// TIA Portal V18 export
ORGANIZATION_BLOCK "Work"   // OB123, LAD, ProgramCycle
TITLE = "Main Program Sweep (Cycle)"
{ S7_Optimized_Access := 'TRUE' }
VERSION : 0.1
// stored: AutoNumber true, IsIECCheckEnabled false, SetENOAutomatically false
   VAR_INPUT
      Initial_Call : Bool;   // Initial call of this OB
      Remanence : Bool;   // =True, if remanent data are available
   END_VAR
BEGIN

REGION Network 1: Active machine
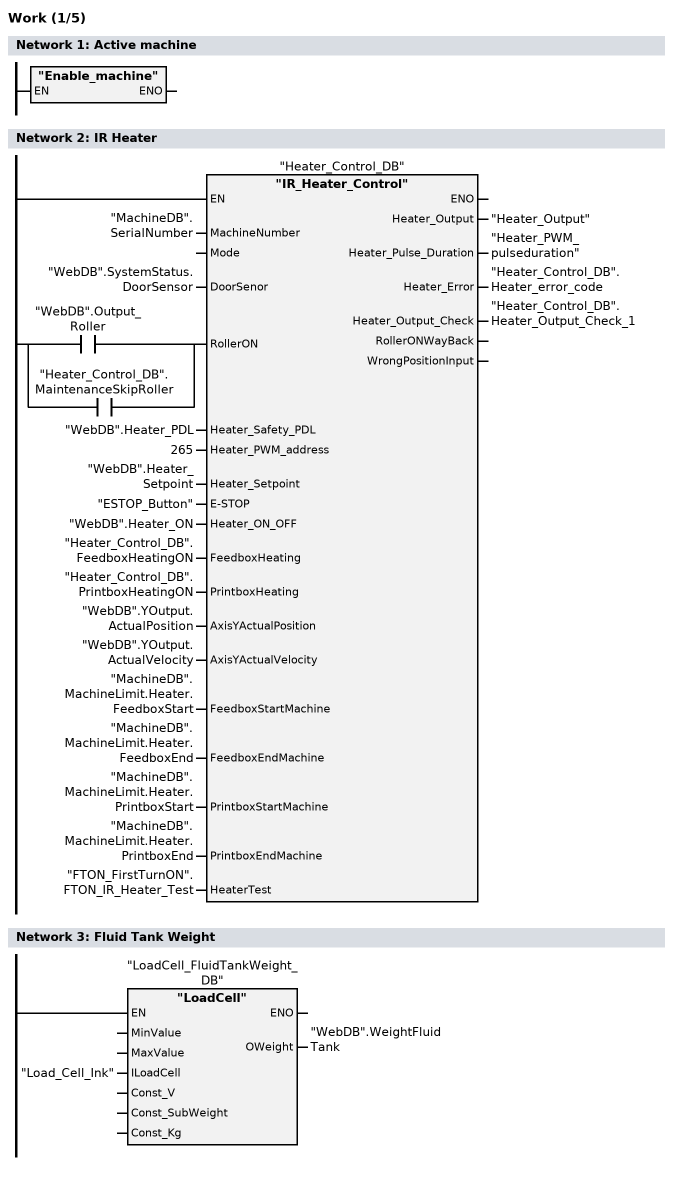
   RUNG wire#powerrail
      "Enable_machine"()
   END_RUNG
   // the same network as SCL:
   "Enable_machine"();
END_REGION

REGION Network 2: IR Heater
   RUNG wire#powerrail
      "Heater_Control_DB"(RollerON := wire#w1, MachineNumber := "MachineDB".SerialNumber, Mode :=, DoorSenor := "WebDB".SystemStatus.DoorSensor, Heater_Safety_PDL := "WebDB".Heater_PDL, Heater_PWM_address := 265, Heater_Setpoint := "WebDB".Heater_Setpoint, "E-STOP" := "ESTOP_Button", Heater_ON_OFF := "WebDB".Heater_ON, FeedboxHeating := "Heater_Control_DB".FeedboxHeatingON, PrintboxHeating := "Heater_Control_DB".PrintboxHeatingON, AxisYActualPosition := "WebDB".YOutput.ActualPosition, AxisYActualVelocity := "WebDB".YOutput.ActualVelocity, FeedboxStartMachine := "MachineDB".MachineLimit.Heater.FeedboxStart, FeedboxEndMachine := "MachineDB".MachineLimit.Heater.FeedboxEnd, PrintboxStartMachine := "MachineDB".MachineLimit.Heater.PrintboxStart, PrintboxEndMachine := "MachineDB".MachineLimit.Heater.PrintboxEnd, HeaterTest := "FTON_FirstTurnON".FTON_IR_Heater_Test, Heater_Output => "Heater_Output", Heater_Pulse_Duration => "Heater_PWM_pulseduration", Heater_Error => "Heater_Control_DB".Heater_error_code, Heater_Output_Check => "Heater_Control_DB".Heater_Output_Check_1, RollerONWayBack =>, WrongPositionInput =>)
   END_RUNG
   RUNG wire#powerrail
      Contact( "WebDB".Output_Roller )
   END_RUNG wire#w1
   RUNG wire#powerrail
      Contact( "Heater_Control_DB".MaintenanceSkipRoller )
   END_RUNG wire#w1
   // the same network as SCL:
   "Heater_Control_DB"(MachineNumber := "MachineDB".SerialNumber,   // "IR_Heater_Control"
                       DoorSenor := "WebDB".SystemStatus.DoorSensor,
                       RollerON := "WebDB".Output_Roller OR "Heater_Control_DB".MaintenanceSkipRoller,
                       Heater_Safety_PDL := "WebDB".Heater_PDL,
                       Heater_PWM_address := 265,
                       Heater_Setpoint := "WebDB".Heater_Setpoint,
                       "E-STOP" := "ESTOP_Button",
                       Heater_ON_OFF := "WebDB".Heater_ON,
                       FeedboxHeating := "Heater_Control_DB".FeedboxHeatingON,
                       PrintboxHeating := "Heater_Control_DB".PrintboxHeatingON,
                       AxisYActualPosition := "WebDB".YOutput.ActualPosition,
                       AxisYActualVelocity := "WebDB".YOutput.ActualVelocity,
                       FeedboxStartMachine := "MachineDB".MachineLimit.Heater.FeedboxStart,
                       FeedboxEndMachine := "MachineDB".MachineLimit.Heater.FeedboxEnd,
                       PrintboxStartMachine := "MachineDB".MachineLimit.Heater.PrintboxStart,
                       PrintboxEndMachine := "MachineDB".MachineLimit.Heater.PrintboxEnd,
                       HeaterTest := "FTON_FirstTurnON".FTON_IR_Heater_Test,
                       Heater_Output => "Heater_Output",
                       Heater_Pulse_Duration => "Heater_PWM_pulseduration",
                       Heater_Error => "Heater_Control_DB".Heater_error_code,
                       Heater_Output_Check => "Heater_Control_DB".Heater_Output_Check_1);
END_REGION

REGION Network 3: Fluid Tank Weight
   RUNG wire#powerrail
      "LoadCell_FluidTankWeight_DB"(MinValue :=, MaxValue :=, ILoadCell := "Load_Cell_Ink", Const_V :=, Const_SubWeight :=, Const_Kg :=, OWeight => "WebDB".WeightFluidTank)
   END_RUNG
   // the same network as SCL:
   "LoadCell_FluidTankWeight_DB"(ILoadCell := "Load_Cell_Ink", OWeight => "WebDB".WeightFluidTank);   // "LoadCell"
END_REGION

REGION Network 4: Fluid Waste Weight
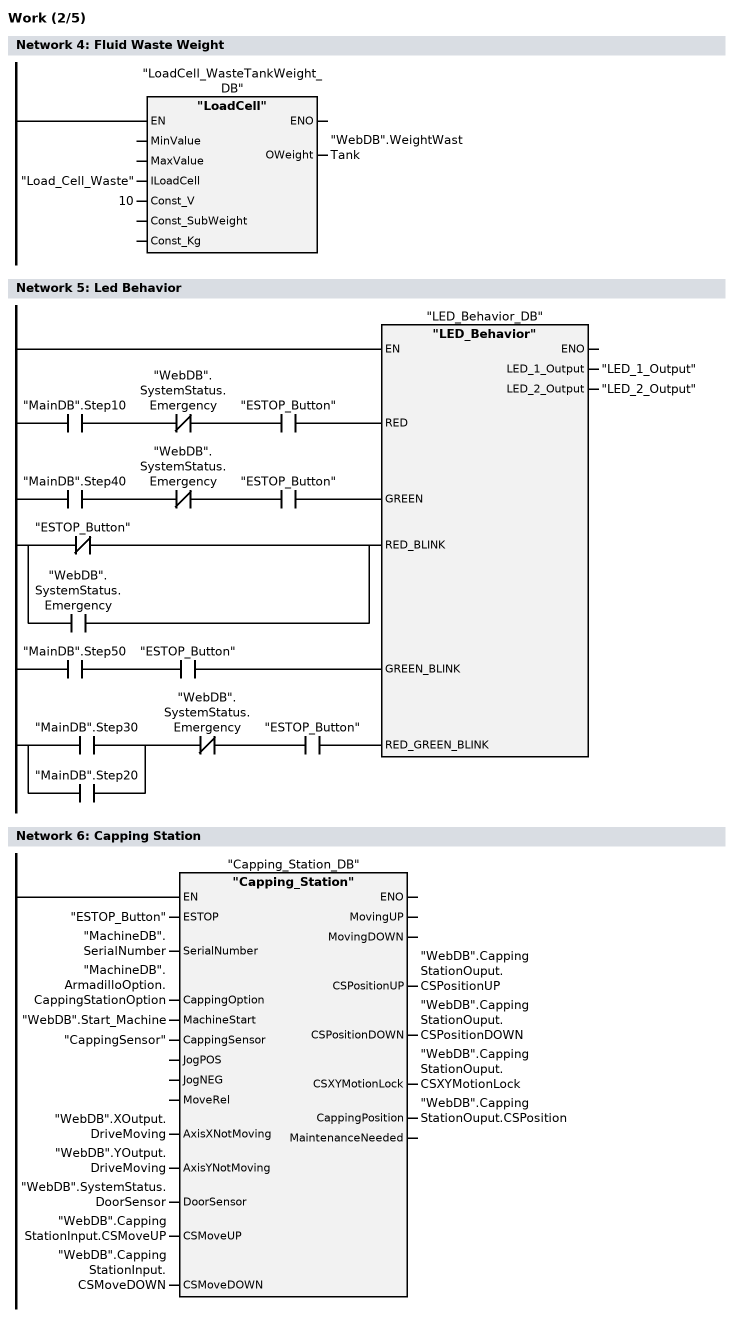
   RUNG wire#powerrail
      "LoadCell_WasteTankWeight_DB"(MinValue :=, MaxValue :=, ILoadCell := "Load_Cell_Waste", Const_V := 10, Const_SubWeight :=, Const_Kg :=, OWeight => "WebDB".WeightWastTank)
   END_RUNG
   // the same network as SCL:
   "LoadCell_WasteTankWeight_DB"(ILoadCell := "Load_Cell_Waste",   // "LoadCell"
                           Const_V := 10,
                           OWeight => "WebDB".WeightWastTank);
END_REGION

REGION Network 5: Led Behavior
   RUNG wire#powerrail
      "LED_Behavior_DB"(RED := wire#w1, GREEN := wire#w2, RED_BLINK := wire#w3, GREEN_BLINK := wire#w4, RED_GREEN_BLINK := wire#w6, LED_1_Output => "LED_1_Output", LED_2_Output => "LED_2_Output")
   END_RUNG
   RUNG wire#powerrail
      Contact( "MainDB".Step10 )
      I_Contact( "WebDB".SystemStatus.Emergency )
      Contact( "ESTOP_Button" )
   END_RUNG wire#w1
   RUNG wire#powerrail
      Contact( "MainDB".Step40 )
      I_Contact( "WebDB".SystemStatus.Emergency )
      Contact( "ESTOP_Button" )
   END_RUNG wire#w2
   RUNG wire#powerrail
      I_Contact( "ESTOP_Button" )
   END_RUNG wire#w3
   RUNG wire#powerrail
      Contact( "WebDB".SystemStatus.Emergency )
   END_RUNG wire#w3
   RUNG wire#powerrail
      Contact( "MainDB".Step50 )
      Contact( "ESTOP_Button" )
   END_RUNG wire#w4
   RUNG wire#powerrail
      Contact( "MainDB".Step30 )
      wire#w5
      I_Contact( "WebDB".SystemStatus.Emergency )
      Contact( "ESTOP_Button" )
   END_RUNG wire#w6
   RUNG wire#powerrail
      Contact( "MainDB".Step20 )
   END_RUNG wire#w5
   // the same network as SCL:
   "LED_Behavior_DB"(RED := "MainDB".Step10 AND NOT "WebDB".SystemStatus.Emergency AND "ESTOP_Button",   // "LED_Behavior"
                     GREEN := "MainDB".Step40 AND NOT "WebDB".SystemStatus.Emergency AND "ESTOP_Button",
                     RED_BLINK := NOT "ESTOP_Button" OR "WebDB".SystemStatus.Emergency,
                     GREEN_BLINK := "MainDB".Step50 AND "ESTOP_Button",
                     RED_GREEN_BLINK := ("MainDB".Step30 OR "MainDB".Step20) AND NOT "WebDB".SystemStatus.Emergency AND "ESTOP_Button",
                     LED_1_Output => "LED_1_Output",
                     LED_2_Output => "LED_2_Output");
END_REGION

REGION Network 6: Capping Station
   RUNG wire#powerrail
      "Capping_Station_DB"(ESTOP := "ESTOP_Button", SerialNumber := "MachineDB".SerialNumber, CappingOption := "MachineDB".ArmadilloOption.CappingStationOption, MachineStart := "WebDB".Start_Machine, CappingSensor := "CappingSensor", JogPOS :=, JogNEG :=, MoveRel :=, AxisXNotMoving := "WebDB".XOutput.DriveMoving, AxisYNotMoving := "WebDB".YOutput.DriveMoving, DoorSensor := "WebDB".SystemStatus.DoorSensor, CSMoveUP := "WebDB".CappingStationInput.CSMoveUP, CSMoveDOWN := "WebDB".CappingStationInput.CSMoveDOWN, MovingUP =>, MovingDOWN =>, CSPositionUP => "WebDB".CappingStationOuput.CSPositionUP, CSPositionDOWN => "WebDB".CappingStationOuput.CSPositionDOWN, CSXYMotionLock => "WebDB".CappingStationOuput.CSXYMotionLock, CappingPosition => "WebDB".CappingStationOuput.CSPosition, MaintenanceNeeded =>)
   END_RUNG
   // the same network as SCL:
   "Capping_Station_DB"(ESTOP := "ESTOP_Button",   // "Capping_Station"
                        SerialNumber := "MachineDB".SerialNumber,
                        CappingOption := "MachineDB".ArmadilloOption.CappingStationOption,
                        MachineStart := "WebDB".Start_Machine,
                        CappingSensor := "CappingSensor",
                        AxisXNotMoving := "WebDB".XOutput.DriveMoving,
                        AxisYNotMoving := "WebDB".YOutput.DriveMoving,
                        DoorSensor := "WebDB".SystemStatus.DoorSensor,
                        CSMoveUP := "WebDB".CappingStationInput.CSMoveUP,
                        CSMoveDOWN := "WebDB".CappingStationInput.CSMoveDOWN,
                        CSPositionUP => "WebDB".CappingStationOuput.CSPositionUP,
                        CSPositionDOWN => "WebDB".CappingStationOuput.CSPositionDOWN,
                        CSXYMotionLock => "WebDB".CappingStationOuput.CSXYMotionLock,
                        CappingPosition => "WebDB".CappingStationOuput.CSPosition);
END_REGION

REGION Network 7: Initial Test Sequence
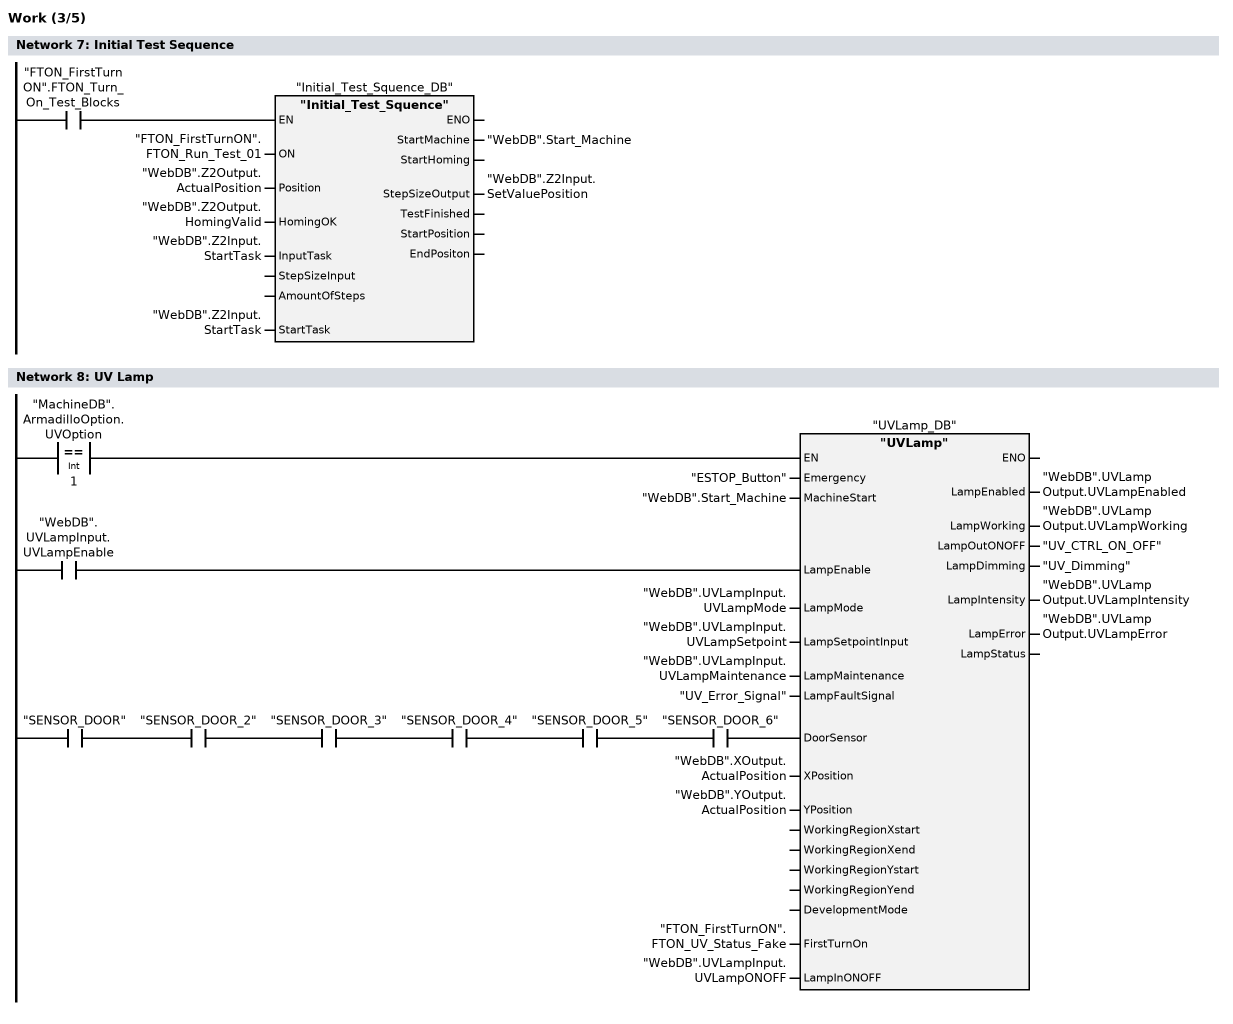
   RUNG wire#powerrail
      Contact( "FTON_FirstTurnON".FTON_Turn_On_Test_Blocks )
      "Initial_Test_Squence_DB"(ON := "FTON_FirstTurnON".FTON_Run_Test_01, Position := "WebDB".Z2Output.ActualPosition, HomingOK := "WebDB".Z2Output.HomingValid, InputTask := "WebDB".Z2Input.StartTask, StepSizeInput :=, AmountOfSteps :=, StartTask := "WebDB".Z2Input.StartTask, StartMachine => "WebDB".Start_Machine, StartHoming =>, StepSizeOutput => "WebDB".Z2Input.SetValuePosition, TestFinished =>, StartPosition =>, EndPositon =>)
   END_RUNG
   // the same network as SCL:
   IF "FTON_FirstTurnON".FTON_Turn_On_Test_Blocks THEN
       "Initial_Test_Squence_DB"(ON := "FTON_FirstTurnON".FTON_Run_Test_01,   // "Initial_Test_Squence"
                               Position := "WebDB".Z2Output.ActualPosition,
                               HomingOK := "WebDB".Z2Output.HomingValid,
                               InputTask := "WebDB".Z2Input.StartTask,
                               StartTask := "WebDB".Z2Input.StartTask,
                               StartMachine => "WebDB".Start_Machine,
                               StepSizeOutput => "WebDB".Z2Input.SetValuePosition);
   END_IF;
END_REGION

REGION Network 8: UV Lamp
   RUNG wire#powerrail
      { S7_Templates := "SrcType := Int" } EQ_Contact(in1 := "MachineDB".ArmadilloOption.UVOption, in2 := 1)
      "UVLamp_DB"(LampEnable := wire#w1, DoorSensor := wire#w2, Emergency := "ESTOP_Button", MachineStart := "WebDB".Start_Machine, LampMode := "WebDB".UVLampInput.UVLampMode, LampSetpointInput := "WebDB".UVLampInput.UVLampSetpoint, LampMaintenance := "WebDB".UVLampInput.UVLampMaintenance, LampFaultSignal := "UV_Error_Signal", XPosition := "WebDB".XOutput.ActualPosition, YPosition := "WebDB".YOutput.ActualPosition, WorkingRegionXstart :=, WorkingRegionXend :=, WorkingRegionYstart :=, WorkingRegionYend :=, DevelopmentMode :=, FirstTurnOn := "FTON_FirstTurnON".FTON_UV_Status_Fake, LampInONOFF := "WebDB".UVLampInput.UVLampONOFF, LampEnabled => "WebDB".UVLampOutput.UVLampEnabled, LampWorking => "WebDB".UVLampOutput.UVLampWorking, LampOutONOFF => "UV_CTRL_ON_OFF", LampDimming => "UV_Dimming", LampIntensity => "WebDB".UVLampOutput.UVLampIntensity, LampError => "WebDB".UVLampOutput.UVLampError, LampStatus =>)
   END_RUNG
   RUNG wire#powerrail
      Contact( "WebDB".UVLampInput.UVLampEnable )
   END_RUNG wire#w1
   RUNG wire#powerrail
      Contact( "SENSOR_DOOR" )
      Contact( "SENSOR_DOOR_2" )
      Contact( "SENSOR_DOOR_3" )
      Contact( "SENSOR_DOOR_4" )
      Contact( "SENSOR_DOOR_5" )
      Contact( "SENSOR_DOOR_6" )
   END_RUNG wire#w2
   // the same network as SCL:
   IF "MachineDB".ArmadilloOption.UVOption = 1 THEN
       "UVLamp_DB"(Emergency := "ESTOP_Button",   // "UVLamp"
                   MachineStart := "WebDB".Start_Machine,
                   LampEnable := "WebDB".UVLampInput.UVLampEnable,
                   LampMode := "WebDB".UVLampInput.UVLampMode,
                   LampSetpointInput := "WebDB".UVLampInput.UVLampSetpoint,
                   LampMaintenance := "WebDB".UVLampInput.UVLampMaintenance,
                   LampFaultSignal := "UV_Error_Signal",
                   DoorSensor := "SENSOR_DOOR" AND "SENSOR_DOOR_2" AND "SENSOR_DOOR_3" AND "SENSOR_DOOR_4" AND "SENSOR_DOOR_5" AND "SENSOR_DOOR_6",
                   XPosition := "WebDB".XOutput.ActualPosition,
                   YPosition := "WebDB".YOutput.ActualPosition,
                   FirstTurnOn := "FTON_FirstTurnON".FTON_UV_Status_Fake,
                   LampInONOFF := "WebDB".UVLampInput.UVLampONOFF,
                   LampEnabled => "WebDB".UVLampOutput.UVLampEnabled,
                   LampWorking => "WebDB".UVLampOutput.UVLampWorking,
                   LampOutONOFF => "UV_CTRL_ON_OFF",
                   LampDimming => "UV_Dimming",
                   LampIntensity => "WebDB".UVLampOutput.UVLampIntensity,
                   LampError => "WebDB".UVLampOutput.UVLampError);
   END_IF;
END_REGION

REGION Network 9: Stacklight
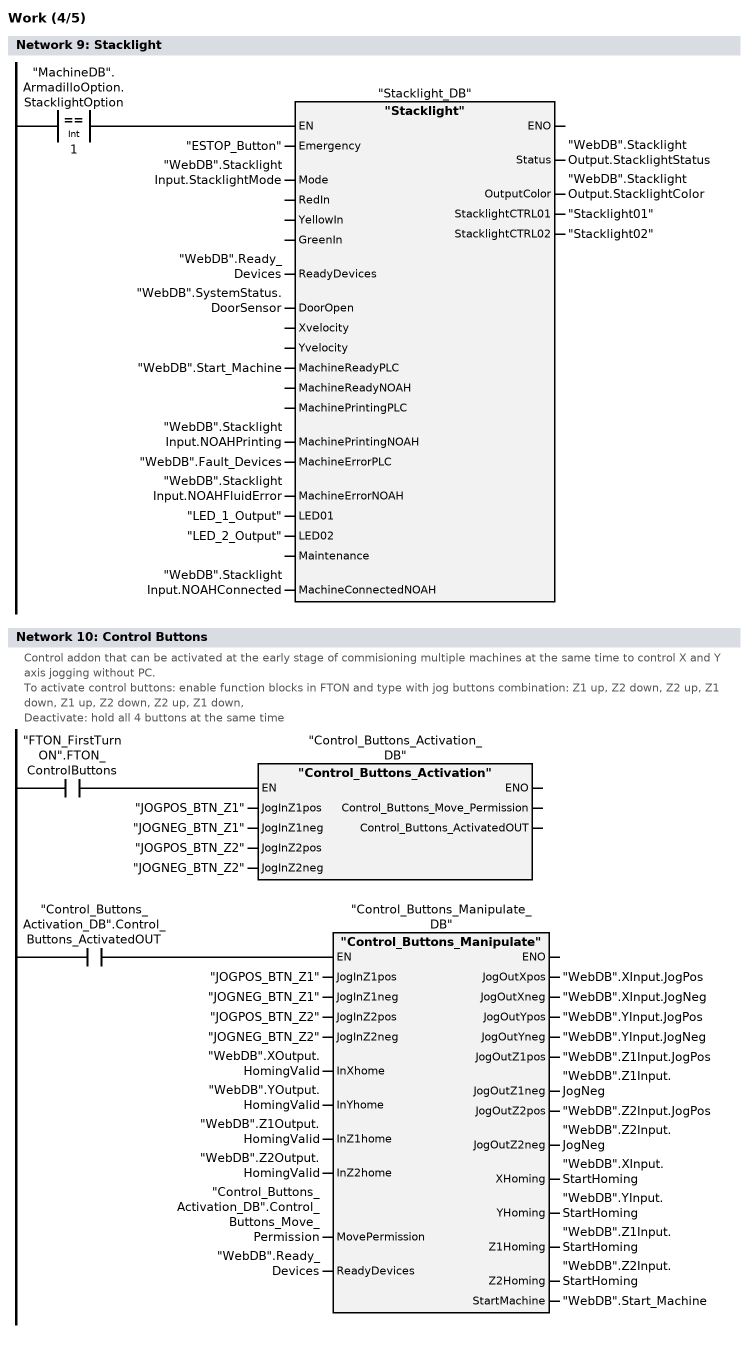
   RUNG wire#powerrail
      { S7_Templates := "SrcType := Int" } EQ_Contact(in1 := "MachineDB".ArmadilloOption.StacklightOption, in2 := 1)
      "Stacklight_DB"(Emergency := "ESTOP_Button", Mode := "WebDB".StacklightInput.StacklightMode, RedIn :=, YellowIn :=, GreenIn :=, ReadyDevices := "WebDB".Ready_Devices, DoorOpen := "WebDB".SystemStatus.DoorSensor, Xvelocity :=, Yvelocity :=, MachineReadyPLC := "WebDB".Start_Machine, MachineReadyNOAH :=, MachinePrintingPLC :=, MachinePrintingNOAH := "WebDB".StacklightInput.NOAHPrinting, MachineErrorPLC := "WebDB".Fault_Devices, MachineErrorNOAH := "WebDB".StacklightInput.NOAHFluidError, LED01 := "LED_1_Output", LED02 := "LED_2_Output", Maintenance :=, MachineConnectedNOAH := "WebDB".StacklightInput.NOAHConnected, Status => "WebDB".StacklightOutput.StacklightStatus, OutputColor => "WebDB".StacklightOutput.StacklightColor, StacklightCTRL01 => "Stacklight01", StacklightCTRL02 => "Stacklight02")
   END_RUNG
   // the same network as SCL:
   IF "MachineDB".ArmadilloOption.StacklightOption = 1 THEN
       "Stacklight_DB"(Emergency := "ESTOP_Button",   // "Stacklight"
                       Mode := "WebDB".StacklightInput.StacklightMode,
                       ReadyDevices := "WebDB".Ready_Devices,
                       DoorOpen := "WebDB".SystemStatus.DoorSensor,
                       MachineReadyPLC := "WebDB".Start_Machine,
                       MachinePrintingNOAH := "WebDB".StacklightInput.NOAHPrinting,
                       MachineErrorPLC := "WebDB".Fault_Devices,
                       MachineErrorNOAH := "WebDB".StacklightInput.NOAHFluidError,
                       LED01 := "LED_1_Output",
                       LED02 := "LED_2_Output",
                       MachineConnectedNOAH := "WebDB".StacklightInput.NOAHConnected,
                       Status => "WebDB".StacklightOutput.StacklightStatus,
                       OutputColor => "WebDB".StacklightOutput.StacklightColor,
                       StacklightCTRL01 => "Stacklight01",
                       StacklightCTRL02 => "Stacklight02");
   END_IF;
END_REGION

REGION Network 10: Control Buttons
   // Control addon that can be activated at the early stage of commisioning multiple machines at the same time to control X and Y axis jogging without PC.
   // 
   // To activate control buttons: enable function blocks in FTON and type with jog buttons combination: Z1 up, Z2 down, Z2 up, Z1 down, Z1 up, Z2 down, Z2 up, Z1 down,
   // 
   // Deactivate: hold all 4 buttons at the same time
   RUNG wire#powerrail
      Contact( "FTON_FirstTurnON".FTON_ControlButtons )
      "Control_Buttons_Activation_DB"(JogInZ1pos := "JOGPOS_BTN_Z1", JogInZ1neg := "JOGNEG_BTN_Z1", JogInZ2pos := "JOGPOS_BTN_Z2", JogInZ2neg := "JOGNEG_BTN_Z2", Control_Buttons_Move_Permission =>, Control_Buttons_ActivatedOUT =>)
   END_RUNG
   RUNG wire#powerrail
      Contact( "Control_Buttons_Activation_DB".Control_Buttons_ActivatedOUT )
      "Control_Buttons_Manipulate_DB"(JogInZ1pos := "JOGPOS_BTN_Z1", JogInZ1neg := "JOGNEG_BTN_Z1", JogInZ2pos := "JOGPOS_BTN_Z2", JogInZ2neg := "JOGNEG_BTN_Z2", InXhome := "WebDB".XOutput.HomingValid, InYhome := "WebDB".YOutput.HomingValid, InZ1home := "WebDB".Z1Output.HomingValid, InZ2home := "WebDB".Z2Output.HomingValid, MovePermission := "Control_Buttons_Activation_DB".Control_Buttons_Move_Permission, ReadyDevices := "WebDB".Ready_Devices, JogOutXpos => "WebDB".XInput.JogPos, JogOutXneg => "WebDB".XInput.JogNeg, JogOutYpos => "WebDB".YInput.JogPos, JogOutYneg => "WebDB".YInput.JogNeg, JogOutZ1pos => "WebDB".Z1Input.JogPos, JogOutZ1neg => "WebDB".Z1Input.JogNeg, JogOutZ2pos => "WebDB".Z2Input.JogPos, JogOutZ2neg => "WebDB".Z2Input.JogNeg, XHoming => "WebDB".XInput.StartHoming, YHoming => "WebDB".YInput.StartHoming, Z1Homing => "WebDB".Z1Input.StartHoming, Z2Homing => "WebDB".Z2Input.StartHoming, StartMachine => "WebDB".Start_Machine)
   END_RUNG
   // the same network as SCL:
   IF "FTON_FirstTurnON".FTON_ControlButtons THEN
       "Control_Buttons_Activation_DB"(JogInZ1pos := "JOGPOS_BTN_Z1",   // "Control_Buttons_Activation"
                               JogInZ1neg := "JOGNEG_BTN_Z1",
                               JogInZ2pos := "JOGPOS_BTN_Z2",
                               JogInZ2neg := "JOGNEG_BTN_Z2");
   END_IF;
   IF "Control_Buttons_Activation_DB".Control_Buttons_ActivatedOUT THEN
       "Control_Buttons_Manipulate_DB"(JogInZ1pos := "JOGPOS_BTN_Z1",   // "Control_Buttons_Manipulate"
                               JogInZ1neg := "JOGNEG_BTN_Z1",
                               JogInZ2pos := "JOGPOS_BTN_Z2",
                               JogInZ2neg := "JOGNEG_BTN_Z2",
                               InXhome := "WebDB".XOutput.HomingValid,
                               InYhome := "WebDB".YOutput.HomingValid,
                               InZ1home := "WebDB".Z1Output.HomingValid,
                               InZ2home := "WebDB".Z2Output.HomingValid,
                               MovePermission := "Control_Buttons_Activation_DB".Control_Buttons_Move_Permission,
                               ReadyDevices := "WebDB".Ready_Devices,
                               JogOutXpos => "WebDB".XInput.JogPos,
                               JogOutXneg => "WebDB".XInput.JogNeg,
                               JogOutYpos => "WebDB".YInput.JogPos,
                               JogOutYneg => "WebDB".YInput.JogNeg,
                               JogOutZ1pos => "WebDB".Z1Input.JogPos,
                               JogOutZ1neg => "WebDB".Z1Input.JogNeg,
                               JogOutZ2pos => "WebDB".Z2Input.JogPos,
                               JogOutZ2neg => "WebDB".Z2Input.JogNeg,
                               XHoming => "WebDB".XInput.StartHoming,
                               YHoming => "WebDB".YInput.StartHoming,
                               Z1Homing => "WebDB".Z1Input.StartHoming,
                               Z2Homing => "WebDB".Z2Input.StartHoming,
                               StartMachine => "WebDB".Start_Machine);
   END_IF;
END_REGION

REGION Network 11: Data Logging
   // Details to start the logging process:
   // 1) Activate web server
   // 2) Set variables to log by assigning them to DataLogging block inputs
   // 3) Create logging file in the FTON
   // 4) Start logging in the FTON
   // 5) Download the file via web server
   // 
   // There is a limited amount of data that can be written due to limited memory capacity. The file will be overwritten after certain amount of records. It is possible to create a new file based on amount of records, should be developed in the future.
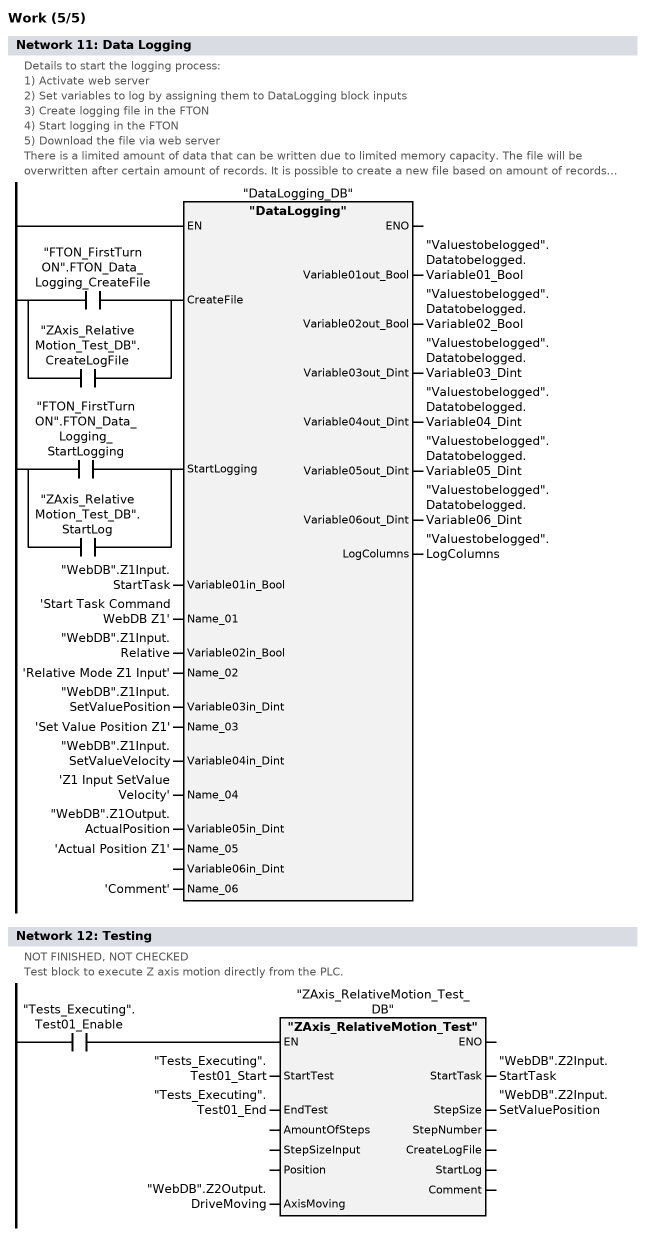
   RUNG wire#powerrail
      "DataLogging_DB"(CreateFile := wire#w1, StartLogging := wire#w2, Variable01in_Bool := "WebDB".Z1Input.StartTask, Name_01 := 'Start Task Command WebDB Z1', Variable02in_Bool := "WebDB".Z1Input.Relative, Name_02 := 'Relative Mode Z1 Input', Variable03in_Dint := "WebDB".Z1Input.SetValuePosition, Name_03 := 'Set Value Position Z1', Variable04in_Dint := "WebDB".Z1Input.SetValueVelocity, Name_04 := 'Z1 Input SetValueVelocity', Variable05in_Dint := "WebDB".Z1Output.ActualPosition, Name_05 := 'Actual Position Z1', Variable06in_Dint :=, Name_06 := 'Comment', Variable01out_Bool => "Valuestobelogged".Datatobelogged.Variable01_Bool, Variable02out_Bool => "Valuestobelogged".Datatobelogged.Variable02_Bool, Variable03out_Dint => "Valuestobelogged".Datatobelogged.Variable03_Dint, Variable04out_Dint => "Valuestobelogged".Datatobelogged.Variable04_Dint, Variable05out_Dint => "Valuestobelogged".Datatobelogged.Variable05_Dint, Variable06out_Dint => "Valuestobelogged".Datatobelogged.Variable06_Dint, LogColumns => "Valuestobelogged".LogColumns)
   END_RUNG
   RUNG wire#powerrail
      Contact( "FTON_FirstTurnON".FTON_Data_Logging_CreateFile )
   END_RUNG wire#w1
   RUNG wire#powerrail
      Contact( "ZAxis_RelativeMotion_Test_DB".CreateLogFile )
   END_RUNG wire#w1
   RUNG wire#powerrail
      Contact( "FTON_FirstTurnON".FTON_Data_Logging_StartLogging )
   END_RUNG wire#w2
   RUNG wire#powerrail
      Contact( "ZAxis_RelativeMotion_Test_DB".StartLog )
   END_RUNG wire#w2
   // the same network as SCL:
   "DataLogging_DB"(CreateFile := "FTON_FirstTurnON".FTON_Data_Logging_CreateFile OR "ZAxis_RelativeMotion_Test_DB".CreateLogFile,   // "DataLogging"
                    StartLogging := "FTON_FirstTurnON".FTON_Data_Logging_StartLogging OR "ZAxis_RelativeMotion_Test_DB".StartLog,
                    Variable01in_Bool := "WebDB".Z1Input.StartTask,
                    Name_01 := 'Start Task Command WebDB Z1',
                    Variable02in_Bool := "WebDB".Z1Input.Relative,
                    Name_02 := 'Relative Mode Z1 Input',
                    Variable03in_Dint := "WebDB".Z1Input.SetValuePosition,
                    Name_03 := 'Set Value Position Z1',
                    Variable04in_Dint := "WebDB".Z1Input.SetValueVelocity,
                    Name_04 := 'Z1 Input SetValueVelocity',
                    Variable05in_Dint := "WebDB".Z1Output.ActualPosition,
                    Name_05 := 'Actual Position Z1',
                    Name_06 := 'Comment',
                    Variable01out_Bool => "Valuestobelogged".Datatobelogged.Variable01_Bool,
                    Variable02out_Bool => "Valuestobelogged".Datatobelogged.Variable02_Bool,
                    Variable03out_Dint => "Valuestobelogged".Datatobelogged.Variable03_Dint,
                    Variable04out_Dint => "Valuestobelogged".Datatobelogged.Variable04_Dint,
                    Variable05out_Dint => "Valuestobelogged".Datatobelogged.Variable05_Dint,
                    Variable06out_Dint => "Valuestobelogged".Datatobelogged.Variable06_Dint,
                    LogColumns => "Valuestobelogged".LogColumns);
END_REGION

REGION Network 12: Testing
   // NOT FINISHED, NOT CHECKED
   // Test block to execute Z axis motion directly from the PLC.
   RUNG wire#powerrail
      Contact( "Tests_Executing".Test01_Enable )
      "ZAxis_RelativeMotion_Test_DB"(StartTest := "Tests_Executing".Test01_Start, EndTest := "Tests_Executing".Test01_End, AmountOfSteps :=, StepSizeInput :=, Position :=, AxisMoving := "WebDB".Z2Output.DriveMoving, StartTask => "WebDB".Z2Input.StartTask, StepSize => "WebDB".Z2Input.SetValuePosition, StepNumber =>, CreateLogFile =>, StartLog =>, Comment =>)
   END_RUNG
   // the same network as SCL:
   IF "Tests_Executing".Test01_Enable THEN
       "ZAxis_RelativeMotion_Test_DB"(StartTest := "Tests_Executing".Test01_Start,   // "ZAxis_RelativeMotion_Test"
                               EndTest := "Tests_Executing".Test01_End,
                               AxisMoving := "WebDB".Z2Output.DriveMoving,
                               StartTask => "WebDB".Z2Input.StartTask,
                               StepSize => "WebDB".Z2Input.SetValuePosition);
   END_IF;
END_REGION
END_ORGANIZATION_BLOCK
